PROGRAM Q10
VAR
	extrude		: BOOL	:= FALSE;
	extruding 	: BOOL 	:= FALSE;
	extruded	: BOOL	:= FALSE;
	warning		: BOOL	:= FALSE;
	TON_0: TON;
	
	count_i		: UINT	:=0;
	count_t		: TIME	:= T#0S;
END_VAR

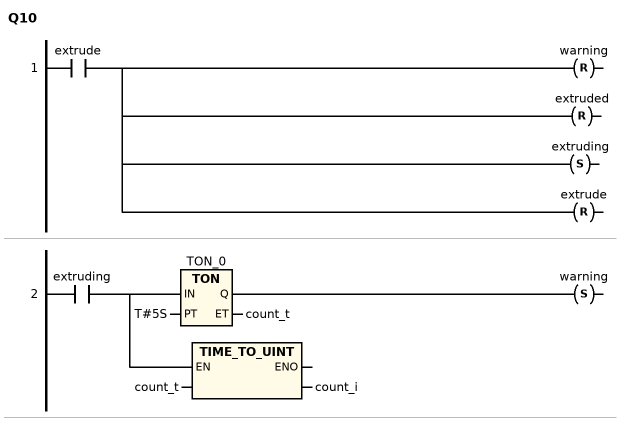
// NETWORK 1
warning R= extrude;
extruded R= extrude;
extruding S= extrude;
extrude R= extrude;

// NETWORK 2
TON_0(IN := extruding, PT := T#5S, ET => count_t); // TON
warning S= TON_0.Q;
IF extruding THEN count_i := TIME_TO_UINT(count_t); END_IF

END_PROGRAM

(* stored: Version 1.1.0.1, ProductVersion 3.1.4024.12
   POU Q10: Id {f53ccd16-c892-431f-a302-796a75deadca}, SpecialFunc None *)
